// TIA Portal V16 export
// export: Created 2023-03-29T11:03:43.0063864Z, ExportSetting WithDefaults, DisplayName Totally Integrated Automation Portal, DisplayVersion V16 Update 6, DisplayName TIA Portal Version Control Interface, DisplayVersion V16 Update 2, DisplayName TIA Portal Openness, DisplayVersion V16 Update 6, DisplayName STEP 7 Professional, DisplayVersion V16 Update 6, DisplayName STEP 7 Safety, DisplayVersion V16, DisplayName WinCC Advanced, DisplayVersion V16 Update 6
DATA_BLOCK "Zmienne_sterujące_zbiorników"   // DB44
{ S7_Optimized_Access := 'FALSE' }
VERSION : 0.1
// stored: AutoNumber true, DBAccessibleFromOPCUA true, IsOnlyStoredInLoadMemory false, IsWriteProtectedInAS false
   VAR
      Zbiornik_1 : Struct
         active_Zb : Bool;   // znacznik aktywnego zbiornika 1= aktywny
         memRisingLevel_min_Zb : Bool;   // pamięc zbocza osiągniecia poziomu minimum w zbiorniku
         memRisingLevel_max_Zb : Bool;   // pamięc zbocza osiągniecia poziomu max w zbiorniku
         isLevelMax_Zb : Bool;   // bit osiągnieia poziomu max w zbiorniku
         isLevelMin_Zb : Bool;   // bit osiągnieia poziomu min w zbiorniku
         isFilling_Zb : Bool;   // bit aktywacji napełniania zbiornika
         isEptying_Zb { ExternalAccessible := 'False'; ExternalVisible := 'False'; ExternalWritable := 'False'} : Bool;   // bit aktywacji przetłaczania
         is_min_float_Zb : Bool;   // sygnał z pływaka minimum
         is_max_float_Zb : Bool;   // sygnał z pływaka max
         ative_Filling : Bool;   // ustawiony jako aktywny do napełniania
         active_Eptying_ : Bool;   // ustawiony jako aktywny do opróżniania
      END_STRUCT;
      Zbiornik_2 : Struct
         active_Zb : Bool;   // znacznik aktywnego zbiornika 1= aktywny
         memRisingLevel_min_Zb : Bool;   // pamięc zbocza osiągniecia poziomu minimum w zbiorniku
         memRisingLevel_max_Zb : Bool;   // pamięc zbocza osiągniecia poziomu max w zbiorniku
         isLevelMax_Zb : Bool;   // bit osiągnieia poziomu max w zbiorniku
         isLevelMin_Zb : Bool;   // bit osiągnieia poziomu min w zbiorniku
         isFilling_Zb : Bool;   // bit aktywacji napełniania zbiornika
         isEptying_Zb { ExternalAccessible := 'False'; ExternalVisible := 'False'; ExternalWritable := 'False'} : Bool;   // bit aktywacji przetłaczania
         is_min_float_Zb : Bool;   // sygnał z pływaka minimum
         is_max_float_Zb : Bool;   // sygnał z pływaka max
         ative_Filling : Bool;   // ustawiony jako aktywny do napełniania
         active_Eptying_ : Bool;   // ustawiony jako aktywny do opróżniania
      END_STRUCT;
      Zbiornik_3 : Struct
         active_Zb : Bool;   // znacznik aktywnego zbiornika 1= aktywny
         memRisingLevel_min_Zb : Bool;   // pamięc zbocza osiągniecia poziomu minimum w zbiorniku
         memRisingLevel_max_Zb : Bool;   // pamięc zbocza osiągniecia poziomu max w zbiorniku
         isLevelMax_Zb : Bool;   // bit osiągnieia poziomu max w zbiorniku
         isLevelMin_Zb : Bool;   // bit osiągnieia poziomu min w zbiorniku
         isFilling_Zb : Bool;   // bit aktywacji napełniania zbiornika
         isEptying_Zb { ExternalAccessible := 'False'; ExternalVisible := 'False'; ExternalWritable := 'False'} : Bool;   // bit aktywacji przetłaczania
         is_min_float_Zb : Bool;   // sygnał z pływaka minimum
         is_max_float_Zb : Bool;   // sygnał z pływaka max
         ative_Filling : Bool;   // ustawiony jako aktywny do napełniania
         active_Eptying_ : Bool;   // ustawiony jako aktywny do opróżniania
      END_STRUCT;
      Zbiornik_4 : Struct
         active_Zb : Bool;   // znacznik aktywnego zbiornika 1= aktywny
         memRisingLevel_min_Zb : Bool;   // pamięc zbocza osiągniecia poziomu minimum w zbiorniku
         memRisingLevel_max_Zb : Bool;   // pamięc zbocza osiągniecia poziomu max w zbiorniku
         isLevelMax_Zb : Bool;   // bit osiągnieia poziomu max w zbiorniku
         isLevelMin_Zb : Bool;   // bit osiągnieia poziomu min w zbiorniku
         isFilling_Zb : Bool;   // bit aktywacji napełniania zbiornika
         isEptying_Zb { ExternalAccessible := 'False'; ExternalVisible := 'False'; ExternalWritable := 'False'} : Bool;   // bit aktywacji przetłaczania
         is_min_float_Zb : Bool;   // sygnał z pływaka minimum
         is_max_float_Zb : Bool;   // sygnał z pływaka max
         ative_Filling : Bool;   // ustawiony jako aktywny do napełniania
         active_Eptying_ : Bool;   // ustawiony jako aktywny do opróżniania
      END_STRUCT;
      out_weekday : Bool;   // bit genetarora tygodniowego
      start_weekday : Bool;   // bit aktywacji pracy tygodniowej zbiorników
      data_sek : Word;   // licznik sekund trybu tygodniowego
      data_hour : DWord;   // licznik godzin trybu tygodniowego
      actOpenZ10 : Bool;   // bit aktywacji przekazania nowej wartości na otwarcie Z10
      actCloseZ10 : Bool;   // bit aktywacji przekazania wartości na zamknięcie [0] Z10
      testowy1 : Int;   // na potrzeby testu
   END_VAR
BEGIN
END_DATA_BLOCK
